LIN {X 0,Y 259.156,Z 1194.159,A -85,B 0,C 180,E1 -3.982,E2 -3.982} C_VEL
LIN {X 0,Y 240.249,Z 1207.459,A -85,B 0,C 180,E1 -6,E2 -6} C_VEL
LIN {X 0,Y 222.253,Z 1218.996,A -85,B 0,C 180,E1 -8.279,E2 -8.279} C_VEL
LIN {X 0,Y 202.836,Z 1230.338,A -85,B 0,C 180,E1 -11.248,E2 -11.248} C_VEL
LIN {X 0,Y 177.97,Z 1243.274,A -85,B 0,C 180,E1 -16.153,E2 -16.153} C_VEL
LIN {X 0,Y 159.555,Z 1251.828,A -85,B 0,C 180,E1 -21.01,E2 -21.01} C_VEL
LIN {X 0,Y 142.486,Z 1259.1,A -85,B 0,C 180,E1 -27.004,E2 -27.004} C_VEL
LIN {X 0,Y 125.055,Z 1266.027,A -85,B 0,C 180,E1 -35.71,E2 -35.71} C_VEL
LIN {X 0,Y 109.97,Z 1271.615,A -85,B 0,C 180,E1 -47.736,E2 -47.736} C_VEL
LIN {X 0,Y 101.633,Z 1274.813,A -85,B 0,C 180,E1 -59.251,E2 -59.251} C_VEL
LIN {X 0,Y 97.319,Z 1276.772,A -85,B 0,C 180,E1 -70.952,E2 -70.952} C_VEL
LIN {X 0,Y 95.995,Z 1277.735,A -85,B 0,C 180,E1 -81.701,E2 -81.701} C_VEL
LIN {X 0,Y 95.905,Z 1278.05,A -85,B 0,C 180,E1 -90.017,E2 -90.017} C_VEL
LIN {X 0,Y 95.996,Z 1277.726,A -85,B 0,C 180,E1 -98.402,E2 -98.402} C_VEL
LIN {X 0,Y 97.638,Z 1276.598,A -85,B 0,C 180,E1 -110.393,E2 -110.393} C_VEL
LIN {X 0,Y 104.256,Z 1273.841,A -85,B 0,C 180,E1 -125.148,E2 -125.148} C_VEL
LIN {X 0,Y 115.973,Z 1269.325,A -85,B 0,C 180,E1 -137.875,E2 -137.875} C_VEL
LIN {X 0,Y 129.201,Z 1264.301,A -85,B 0,C 180,E1 -146.72,E2 -146.72} C_VEL
LIN {X 0,Y 144.01,Z 1258.396,A -85,B 0,C 180,E1 -153.617,E2 -153.617} C_VEL
LIN {X 0,Y 161.221,Z 1251.006,A -85,B 0,C 180,E1 -159.494,E2 -159.494} C_VEL
LIN {X 0,Y 184.211,Z 1240.12,A -85,B 0,C 180,E1 -165.22,E2 -165.22} C_VEL
LIN {X 0,Y 204.707,Z 1229.147,A -85,B 0,C 180,E1 -169.075,E2 -169.075} C_VEL
LIN {X 0,Y 222.303,Z 1218.82,A -85,B 0,C 180,E1 -171.735,E2 -171.735} C_VEL
LIN {X 0,Y 240.473,Z 1207.142,A -85,B 0,C 180,E1 -174.033,E2 -174.033} C_VEL
LIN {X 0,Y 260.572,Z 1192.942,A -85,B 0,C 180,E1 -176.162,E2 -176.162} C_VEL
LIN {X 0,Y 283.358,Z 1174.812,A -85,B 0,C 180,E1 -178.18,E2 -178.18} C_VEL
LIN {X 0,Y 299.995,Z 1160.095,A -85,B 0,C 180,E1 -179.448,E2 -179.448} C_VEL
LIN {X 0,Y 311.22,Z 1149.435,A -85,B 0,C 180,E1 -180.208,E2 -180.208} C_VEL
LIN {X 0,Y 290.116,Z 1168.891,A -85,B 0,C 180,E1 -181.735,E2 -181.735} C_VEL
LIN {X 0,Y 272.413,Z 1183.527,A -85,B 0,C 180,E1 -183.212,E2 -183.212} C_VEL
LIN {X 0,Y 254.915,Z 1196.706,A -85,B 0,C 180,E1 -184.887,E2 -184.887} C_VEL
LIN {X 0,Y 236.716,Z 1209.198,A -85,B 0,C 180,E1 -186.921,E2 -186.921} C_VEL
LIN {X 0,Y 214.231,Z 1223.155,A -85,B 0,C 180,E1 -189.971,E2 -189.971} C_VEL
LIN {X 0,Y 192.466,Z 1235.016,A -85,B 0,C 180,E1 -193.689,E2 -193.689} C_VEL
LIN {X 0,Y 175.049,Z 1243.639,A -85,B 0,C 180,E1 -197.44,E2 -197.44} C_VEL
LIN {X 0,Y 157.697,Z 1251.486,A -85,B 0,C 180,E1 -202.201,E2 -202.201} C_VEL
LIN {X 0,Y 139.436,Z 1259.064,A -85,B 0,C 180,E1 -208.953,E2 -208.953} C_VEL
LIN {X 0,Y 121.037,Z 1265.976,A -85,B 0,C 180,E1 -219.037,E2 -219.037} C_VEL
LIN {X 0,Y 109.576,Z 1270.085,A -85,B 0,C 180,E1 -228.91,E2 -228.91} C_VEL
LIN {X 0,Y 101.75,Z 1272.968,A -85,B 0,C 180,E1 -239.905,E2 -239.905} C_VEL
LIN {X 0,Y 97.45,Z 1274.785,A -85,B 0,C 180,E1 -251.436,E2 -251.436} C_VEL
LIN {X 0,Y 96.054,Z 1275.667,A -85,B 0,C 180,E1 -262.206,E2 -262.206} C_VEL
LIN {X 0,Y 95.898,Z 1275.918,A -85,B 0,C 180,E1 -271.178,E2 -271.178} C_VEL
LIN {X 0,Y 96.228,Z 1275.57,A -85,B 0,C 180,E1 -280.762,E2 -280.762} C_VEL
LIN {X 0,Y 99.154,Z 1274.127,A -85,B 0,C 180,E1 -294.402,E2 -294.402} C_VEL
LIN {X 0,Y 107.15,Z 1271.002,A -85,B 0,C 180,E1 -308.384,E2 -308.384} C_VEL
LIN {X 0,Y 117.511,Z 1267.28,A -85,B 0,C 180,E1 -318.461,E2 -318.461} C_VEL
LIN {X 0,Y 130.322,Z 1262.576,A -85,B 0,C 180,E1 -326.724,E2 -326.724} C_VEL
LIN {X 0,Y 145.941,Z 1256.491,A -85,B 0,C 180,E1 -333.803,E2 -333.803} C_VEL
LIN {X 0,Y 166.537,Z 1247.783,A -85,B 0,C 180,E1 -340.461,E2 -340.461} C_VEL
LIN {X 0,Y 188.109,Z 1237.371,A -85,B 0,C 180,E1 -345.533,E2 -345.533} C_VEL
LIN {X 0,Y 206.779,Z 1227.428,A -85,B 0,C 180,E1 -348.941,E2 -348.941} C_VEL
LIN {X 0,Y 225.299,Z 1216.585,A -85,B 0,C 180,E1 -351.693,E2 -351.693} C_VEL
LIN {X 0,Y 247.131,Z 1202.487,A -85,B 0,C 180,E1 -354.353,E2 -354.353} C_VEL
LIN {X 0,Y 268.428,Z 1186.87,A -85,B 0,C 180,E1 -356.504,E2 -356.504} C_VEL
LIN {X 0,Y 286.095,Z 1172.556,A -85,B 0,C 180,E1 -358.03,E2 -358.03} C_VEL
LIN {X 0,Y 302.945,Z 1157.563,A -85,B 0,C 180,E1 -359.306,E2 -359.306} C_VEL
LIN {X 0,Y 310.594,Z 1150.361,A -85,B 0,C 180,E1 -359.845,E2 -359.845} C_VEL
LIN {X 0,Y 300.565,Z 1159.826,A -85,B 0,C 180,E1 -360.522,E2 -360.522} C_VEL
LIN {X 0,Y 294.883,Z 1165.108,A -85,B 0,C 180,E1 -360.731,E2 -360.731} C_VEL
LIN {X 0,Y 278.673,Z 1178.812,A -85,B 0,C 180,E1 -360.644,E2 -360.644} C_VEL
LIN {X 0,Y 273.535,Z 1182.795,A -85,B 0,C 180,E1 -360.881,E2 -360.881} C_VEL
LIN {X 0,Y 256.149,Z 1195.901,A -85,B 0,C 180,E1 -362.366,E2 -362.366} C_VEL
LIN {X 0,Y 238.547,Z 1208.008,A -85,B 0,C 180,E1 -364.111,E2 -364.111} C_VEL
LIN {X 0,Y 220.169,Z 1219.529,A -85,B 0,C 180,E1 -366.257,E2 -366.257} C_VEL
LIN {X 0,Y 197.647,Z 1232.322,A -85,B 0,C 180,E1 -369.493,E2 -369.493} C_VEL
LIN {X 0,Y 174.924,Z 1243.592,A -85,B 0,C 180,E1 -373.705,E2 -373.705} C_VEL
LIN {X 0,Y 156.208,Z 1251.959,A -85,B 0,C 180,E1 -378.279,E2 -378.279} C_VEL
LIN {X 0,Y 138.868,Z 1259.009,A -85,B 0,C 180,E1 -383.91,E2 -383.91} C_VEL
LIN {X 0,Y 120.629,Z 1265.829,A -85,B 0,C 180,E1 -392.307,E2 -392.307} C_VEL
LIN {X 0,Y 103.957,Z 1271.525,A -85,B 0,C 180,E1 -404.647,E2 -404.647} C_VEL
LIN {X 0,Y 94.627,Z 1274.723,A -85,B 0,C 180,E1 -416.692,E2 -416.692} C_VEL
LIN {X 0,Y 89.669,Z 1276.668,A -85,B 0,C 180,E1 -429.115,E2 -429.115} C_VEL
LIN {X 0,Y 88.018,Z 1277.644,A -85,B 0,C 180,E1 -440.868,E2 -440.868} C_VEL
LIN {X 0,Y 87.904,Z 1277.963,A -85,B 0,C 180,E1 -450.019,E2 -450.019} C_VEL
LIN {X 0,Y 88.019,Z 1277.638,A -85,B 0,C 180,E1 -459.17,E2 -459.17} C_VEL
LIN {X 0,Y 89.841,Z 1276.578,A -85,B 0,C 180,E1 -471.566,E2 -471.566} C_VEL
LIN {X 0,Y 96.126,Z 1274.204,A -85,B 0,C 180,E1 -485.772,E2 -485.772} C_VEL
LIN {X 0,Y 109.486,Z 1269.616,A -85,B 0,C 180,E1 -500.262,E2 -500.262} C_VEL
LIN {X 0,Y 124.095,Z 1264.466,A -85,B 0,C 180,E1 -509.58,E2 -509.58} C_VEL
LIN {X 0,Y 139.687,Z 1258.61,A -85,B 0,C 180,E1 -516.404,E2 -516.404} C_VEL
LIN {X 0,Y 156.776,Z 1251.627,A -85,B 0,C 180,E1 -521.885,E2 -521.885} C_VEL
LIN {X 0,Y 176.754,Z 1242.649,A -85,B 0,C 180,E1 -526.683,E2 -526.683} C_VEL
LIN {X 0,Y 201.696,Z 1229.933,A -85,B 0,C 180,E1 -531.16,E2 -531.16} C_VEL
LIN {X 0,Y 221.251,Z 1218.726,A -85,B 0,C 180,E1 -533.889,E2 -533.889} C_VEL
LIN {X 0,Y 239.573,Z 1207.163,A -85,B 0,C 180,E1 -536.006,E2 -536.006} C_VEL
LIN {X 0,Y 258.174,Z 1194.258,A -85,B 0,C 180,E1 -537.823,E2 -537.823} C_VEL
LIN {X 0,Y 280.988,Z 1176.612,A -85,B 0,C 180,E1 -539.696,E2 -539.696} C_VEL
LIN {X 0,Y 288.217,Z 1170.471,A -85,B 0,C 180,E1 -540.226,E2 -540.226} C_VEL
LIN {X 0,Y 271.084,Z 1184.386,A -85,B 0,C 180,E1 -541.547,E2 -541.547} C_VEL
LIN {X 0,Y 253.362,Z 1197.496,A -85,B 0,C 180,E1 -543.111,E2 -543.111} C_VEL
LIN {X 0,Y 232.002,Z 1211.815,A -85,B 0,C 180,E1 -545.348,E2 -545.348} C_VEL
LIN {X 0,Y 208.24,Z 1225.801,A -85,B 0,C 180,E1 -548.419,E2 -548.419} C_VEL
LIN {X 0,Y 189.744,Z 1235.564,A -85,B 0,C 180,E1 -551.402,E2 -551.402} C_VEL
LIN {X 0,Y 171.842,Z 1244.133,A -85,B 0,C 180,E1 -554.98,E2 -554.98} C_VEL
LIN {X 0,Y 153.065,Z 1252.278,A -85,B 0,C 180,E1 -559.812,E2 -559.812} C_VEL
LIN {X 0,Y 131.097,Z 1260.81,A -85,B 0,C 180,E1 -567.758,E2 -567.758} C_VEL
LIN {X 0,Y 114.712,Z 1266.474,A -85,B 0,C 180,E1 -576.666,E2 -576.666} C_VEL
LIN {X 0,Y 102.983,Z 1270.333,A -85,B 0,C 180,E1 -586.401,E2 -586.401} C_VEL
LIN {X 0,Y 94.394,Z 1273.169,A -85,B 0,C 180,E1 -598,E2 -598} C_VEL
LIN {X 0,Y 89.607,Z 1274.94,A -85,B 0,C 180,E1 -610.424,E2 -610.424} C_VEL
LIN {X 0,Y 88.053,Z 1275.777,A -85,B 0,C 180,E1 -622.15,E2 -622.15} C_VEL
LIN {X 0,Y 87.899,Z 1276.006,A -85,B 0,C 180,E1 -631.285,E2 -631.285} C_VEL
LIN {X 0,Y 88.245,Z 1275.68,A -85,B 0,C 180,E1 -641.086,E2 -641.086} C_VEL
LIN {X 0,Y 91.516,Z 1274.31,A -85,B 0,C 180,E1 -655.893,E2 -655.893} C_VEL
LIN {X 0,Y 100.534,Z 1271.182,A -85,B 0,C 180,E1 -671.003,E2 -671.003} C_VEL
LIN {X 0,Y 112.164,Z 1267.37,A -85,B 0,C 180,E1 -681.645,E2 -681.645} C_VEL
LIN {X 0,Y 126.259,Z 1262.549,A -85,B 0,C 180,E1 -690.071,E2 -690.071} C_VEL
LIN {X 0,Y 142.567,Z 1256.533,A -85,B 0,C 180,E1 -696.874,E2 -696.874} C_VEL
LIN {X 0,Y 163.922,Z 1247.874,A -85,B 0,C 180,E1 -703.224,E2 -703.224} C_VEL
LIN {X 0,Y 186.01,Z 1237.553,A -85,B 0,C 180,E1 -707.995,E2 -707.995} C_VEL
LIN {X 0,Y 205.337,Z 1227.518,A -85,B 0,C 180,E1 -711.235,E2 -711.235} C_VEL
LIN {X 0,Y 223.289,Z 1217.244,A -85,B 0,C 180,E1 -713.688,E2 -713.688} C_VEL
LIN {X 0,Y 242.557,Z 1205.1,A -85,B 0,C 180,E1 -715.888,E2 -715.888} C_VEL
LIN {X 0,Y 267.061,Z 1187.725,A -85,B 0,C 180,E1 -718.193,E2 -718.193} C_VEL
LIN {X 0,Y 284.932,Z 1173.485,A -85,B 0,C 180,E1 -719.615,E2 -719.615} C_VEL
LIN {X 0,Y 287.634,Z 1171.208,A -85,B 0,C 180,E1 -719.826,E2 -719.826} C_VEL
LIN {X 0,Y 273.535,Z 1182.795,A -85,B 0,C 180,E1 -720.881,E2 -720.881} C_VEL
LIN {X 0,Y 267.462,Z 1187.511,A -85,B 0,C 180,E1 -721.15,E2 -721.15} C_VEL
LIN {X 0,Y 250.268,Z 1199.952,A -85,B 0,C 180,E1 -721.16,E2 -721.16} C_VEL
LIN {X 0,Y 244.838,Z 1203.559,A -85,B 0,C 180,E1 -721.463,E2 -721.463} C_VEL
LIN {X 0,Y 223.382,Z 1217.085,A -85,B 0,C 180,E1 -723.621,E2 -723.621} C_VEL
LIN {X 0,Y 204.053,Z 1228.083,A -85,B 0,C 180,E1 -725.99,E2 -725.99} C_VEL
LIN {X 0,Y 184.206,Z 1238.279,A -85,B 0,C 180,E1 -728.992,E2 -728.992} C_VEL
LIN {X 0,Y 160.383,Z 1249.194,A -85,B 0,C 180,E1 -733.704,E2 -733.704} C_VEL
LIN {X 0,Y 138.962,Z 1257.691,A -85,B 0,C 180,E1 -739.551,E2 -739.551} C_VEL
LIN {X 0,Y 121.526,Z 1263.934,A -85,B 0,C 180,E1 -746.293,E2 -746.293} C_VEL
LIN {X 0,Y 105.71,Z 1269.123,A -85,B 0,C 180,E1 -755.239,E2 -755.239} C_VEL
LIN {X 0,Y 90.657,Z 1273.835,A -85,B 0,C 180,E1 -769.555,E2 -769.555} C_VEL
LIN {X 0,Y 82.633,Z 1276.386,A -85,B 0,C 180,E1 -785.167,E2 -785.167} C_VEL
LIN {X 0,Y 80.099,Z 1277.532,A -85,B 0,C 180,E1 -799.229,E2 -799.229} C_VEL
LIN {X 0,Y 79.896,Z 1277.863,A -85,B 0,C 180,E1 -809.304,E2 -809.304} C_VEL
LIN {X 0,Y 80.001,Z 1277.598,A -85,B 0,C 180,E1 -818.646,E2 -818.646} C_VEL
LIN {X 0,Y 81.557,Z 1276.77,A -85,B 0,C 180,E1 -830.847,E2 -830.847} C_VEL
LIN {X 0,Y 86.413,Z 1275.065,A -85,B 0,C 180,E1 -843.76,E2 -843.76} C_VEL
LIN {X 0,Y 95.914,Z 1272.105,A -85,B 0,C 180,E1 -856.525,E2 -856.525} C_VEL
LIN {X 0,Y 108.767,Z 1268.092,A -85,B 0,C 180,E1 -866.802,E2 -866.802} C_VEL
LIN {X 0,Y 126.154,Z 1262.31,A -85,B 0,C 180,E1 -875.737,E2 -875.737} C_VEL
LIN {X 0,Y 149.161,Z 1253.675,A -85,B 0,C 180,E1 -883.483,E2 -883.483} C_VEL
LIN {X 0,Y 168.619,Z 1245.417,A -85,B 0,C 180,E1 -888.112,E2 -888.112} C_VEL
LIN {X 0,Y 187.058,Z 1236.748,A -85,B 0,C 180,E1 -891.492,E2 -891.492} C_VEL
LIN {X 0,Y 206.022,Z 1226.885,A -85,B 0,C 180,E1 -894.281,E2 -894.281} C_VEL
LIN {X 0,Y 229.302,Z 1213.436,A -85,B 0,C 180,E1 -897.023,E2 -897.023} C_VEL
LIN {X 0,Y 252.014,Z 1198.391,A -85,B 0,C 180,E1 -899.182,E2 -899.182} C_VEL
LIN {X 0,Y 264.989,Z 1189.078,A -85,B 0,C 180,E1 -900.257,E2 -900.257} C_VEL
LIN {X 0,Y 242.172,Z 1204.967,A -85,B 0,C 180,E1 -902.219,E2 -902.219} C_VEL
LIN {X 0,Y 222.604,Z 1217.133,A -85,B 0,C 180,E1 -904.244,E2 -904.244} C_VEL
LIN {X 0,Y 204.315,Z 1227.427,A -85,B 0,C 180,E1 -906.513,E2 -906.513} C_VEL
LIN {X 0,Y 185.471,Z 1237.022,A -85,B 0,C 180,E1 -909.365,E2 -909.365} C_VEL
LIN {X 0,Y 162.144,Z 1247.681,A -85,B 0,C 180,E1 -913.916,E2 -913.916} C_VEL
LIN {X 0,Y 139.459,Z 1256.554,A -85,B 0,C 180,E1 -920.049,E2 -920.049} C_VEL
LIN {X 0,Y 122.809,Z 1262.407,A -85,B 0,C 180,E1 -926.39,E2 -926.39} C_VEL
LIN {X 0,Y 107.947,Z 1267.175,A -85,B 0,C 180,E1 -934.45,E2 -934.45} C_VEL
LIN {X 0,Y 95.035,Z 1271.05,A -85,B 0,C 180,E1 -945.155,E2 -945.155} C_VEL
LIN {X 0,Y 84.858,Z 1274.147,A -85,B 0,C 180,E1 -960.317,E2 -960.317} C_VEL
LIN {X 0,Y 80.485,Z 1275.717,A -85,B 0,C 180,E1 -976.326,E2 -976.326} C_VEL
LIN {X 0,Y 79.919,Z 1276.039,A -85,B 0,C 180,E1 -987.111,E2 -987.111} C_VEL
LIN {X 0,Y 79.987,Z 1275.939,A -85,B 0,C 180,E1 -996.439,E2 -996.439} C_VEL
LIN {X 0,Y 81.441,Z 1275.255,A -85,B 0,C 180,E1 -1009.337,E2 -1009.337} C_VEL
LIN {X 0,Y 86.743,Z 1273.528,A -85,B 0,C 180,E1 -1023.569,E2 -1023.569} C_VEL
LIN {X 0,Y 95.995,Z 1270.802,A -85,B 0,C 180,E1 -1035.92,E2 -1035.92} C_VEL
LIN {X 0,Y 108.508,Z 1267.054,A -85,B 0,C 180,E1 -1045.999,E2 -1045.999} C_VEL
LIN {X 0,Y 124.225,Z 1262.004,A -85,B 0,C 180,E1 -1054.318,E2 -1054.318} C_VEL
LIN {X 0,Y 146.064,Z 1254.251,A -85,B 0,C 180,E1 -1062.058,E2 -1062.058} C_VEL
LIN {X 0,Y 167.963,Z 1245.182,A -85,B 0,C 180,E1 -1067.443,E2 -1067.443} C_VEL
LIN {X 0,Y 187.239,Z 1236.278,A -85,B 0,C 180,E1 -1071.015,E2 -1071.015} C_VEL
LIN {X 0,Y 206.694,Z 1226.289,A -85,B 0,C 180,E1 -1073.891,E2 -1073.891} C_VEL
LIN {X 0,Y 230.321,Z 1212.76,A -85,B 0,C 180,E1 -1076.681,E2 -1076.681} C_VEL
LIN {X 0,Y 253.236,Z 1197.657,A -85,B 0,C 180,E1 -1078.869,E2 -1078.869} C_VEL
LIN {X 0,Y 264.571,Z 1189.623,A -85,B 0,C 180,E1 -1079.81,E2 -1079.81} C_VEL
LIN {X 0,Y 244.838,Z 1203.559,A -85,B 0,C 180,E1 -1081.463,E2 -1081.463} C_VEL
LIN {X 0,Y 238.395,Z 1207.737,A -85,B 0,C 180,E1 -1081.813,E2 -1081.813} C_VEL
LIN {X 0,Y 221.173,Z 1218.143,A -85,B 0,C 180,E1 -1081.931,E2 -1081.931} C_VEL
LIN {X 0,Y 214.631,Z 1221.892,A -85,B 0,C 180,E1 -1082.349,E2 -1082.349} C_VEL
LIN {X 0,Y 189.509,Z 1235.084,A -85,B 0,C 180,E1 -1085.45,E2 -1085.45} C_VEL
LIN {X 0,Y 169.841,Z 1244.228,A -85,B 0,C 180,E1 -1088.571,E2 -1088.571} C_VEL
LIN {X 0,Y 150.526,Z 1252.269,A -85,B 0,C 180,E1 -1092.518,E2 -1092.518} C_VEL
LIN {X 0,Y 130.389,Z 1259.747,A -85,B 0,C 180,E1 -1098.079,E2 -1098.079} C_VEL
LIN {X 0,Y 107.164,Z 1267.258,A -85,B 0,C 180,E1 -1107.809,E2 -1107.809} C_VEL
LIN {X 0,Y 91.737,Z 1271.681,A -85,B 0,C 180,E1 -1118.409,E2 -1118.409} C_VEL
LIN {X 0,Y 80.612,Z 1274.736,A -85,B 0,C 180,E1 -1131.392,E2 -1131.392} C_VEL
LIN {X 0,Y 74.378,Z 1276.56,A -85,B 0,C 180,E1 -1145.396,E2 -1145.396} C_VEL
LIN {X 0,Y 72.115,Z 1277.468,A -85,B 0,C 180,E1 -1158.831,E2 -1158.831} C_VEL
LIN {X 0,Y 71.896,Z 1277.775,A -85,B 0,C 180,E1 -1169.226,E2 -1169.226} C_VEL
LIN {X 0,Y 72.031,Z 1277.509,A -85,B 0,C 180,E1 -1179.612,E2 -1179.612} C_VEL
LIN {X 0,Y 74.024,Z 1276.663,A -85,B 0,C 180,E1 -1193.289,E2 -1193.289} C_VEL
LIN {X 0,Y 80.081,Z 1274.857,A -85,B 0,C 180,E1 -1207.745,E2 -1207.745} C_VEL
LIN {X 0,Y 90.63,Z 1271.946,A -85,B 0,C 180,E1 -1220.585,E2 -1220.585} C_VEL
LIN {X 0,Y 105.139,Z 1267.789,A -85,B 0,C 180,E1 -1231.064,E2 -1231.064} C_VEL
LIN {X 0,Y 126.244,Z 1261.179,A -85,B 0,C 180,E1 -1240.51,E2 -1240.51} C_VEL
LIN {X 0,Y 148.776,Z 1252.868,A -85,B 0,C 180,E1 -1247.073,E2 -1247.073} C_VEL
LIN {X 0,Y 168.021,Z 1244.915,A -85,B 0,C 180,E1 -1251.109,E2 -1251.109} C_VEL
LIN {X 0,Y 186.958,Z 1236.192,A -85,B 0,C 180,E1 -1254.195,E2 -1254.195} C_VEL
LIN {X 0,Y 207.31,Z 1225.754,A -85,B 0,C 180,E1 -1256.843,E2 -1256.843} C_VEL
LIN {X 0,Y 233.276,Z 1210.634,A -85,B 0,C 180,E1 -1259.509,E2 -1259.509} C_VEL
LIN {X 0,Y 241.697,Z 1205.247,A -85,B 0,C 180,E1 -1260.273,E2 -1260.273} C_VEL
LIN {X 0,Y 222.142,Z 1217.226,A -85,B 0,C 180,E1 -1262.095,E2 -1262.095} C_VEL
LIN {X 0,Y 202.996,Z 1227.804,A -85,B 0,C 180,E1 -1264.237,E2 -1264.237} C_VEL
LIN {X 0,Y 183.342,Z 1237.569,A -85,B 0,C 180,E1 -1266.937,E2 -1266.937} C_VEL
LIN {X 0,Y 159.07,Z 1248.271,A -85,B 0,C 180,E1 -1271.268,E2 -1271.268} C_VEL
LIN {X 0,Y 136.81,Z 1256.646,A -85,B 0,C 180,E1 -1276.747,E2 -1276.747} C_VEL
LIN {X 0,Y 119.33,Z 1262.499,A -85,B 0,C 180,E1 -1282.794,E2 -1282.794} C_VEL
LIN {X 0,Y 102.759,Z 1267.47,A -85,B 0,C 180,E1 -1291.072,E2 -1291.072} C_VEL
LIN {X 0,Y 87.523,Z 1271.657,A -85,B 0,C 180,E1 -1303.272,E2 -1303.272} C_VEL
LIN {X 0,Y 76.23,Z 1274.659,A -85,B 0,C 180,E1 -1320.943,E2 -1320.943} C_VEL
LIN {X 0,Y 72.367,Z 1275.868,A -85,B 0,C 180,E1 -1337.205,E2 -1337.205} C_VEL
LIN {X 0,Y 71.907,Z 1276.172,A -85,B 0,C 180,E1 -1348.383,E2 -1348.383} C_VEL
LIN {X 0,Y 72.085,Z 1275.984,A -85,B 0,C 180,E1 -1358.753,E2 -1358.753} C_VEL
LIN {X 0,Y 74.001,Z 1275.278,A -85,B 0,C 180,E1 -1372.205,E2 -1372.205} C_VEL
LIN {X 0,Y 80.096,Z 1273.595,A -85,B 0,C 180,E1 -1386.969,E2 -1386.969} C_VEL
LIN {X 0,Y 91.016,Z 1270.735,A -85,B 0,C 180,E1 -1400.233,E2 -1400.233} C_VEL
LIN {X 0,Y 105.514,Z 1266.738,A -85,B 0,C 180,E1 -1410.634,E2 -1410.634} C_VEL
LIN {X 0,Y 124.909,Z 1260.841,A -85,B 0,C 180,E1 -1419.44,E2 -1419.44} C_VEL
LIN {X 0,Y 148.13,Z 1252.598,A -85,B 0,C 180,E1 -1426.353,E2 -1426.353} C_VEL
LIN {X 0,Y 168.196,Z 1244.47,A -85,B 0,C 180,E1 -1430.615,E2 -1430.615} C_VEL
LIN {X 0,Y 187.068,Z 1235.914,A -85,B 0,C 180,E1 -1433.709,E2 -1433.709} C_VEL
LIN {X 0,Y 208.33,Z 1225.144,A -85,B 0,C 180,E1 -1436.485,E2 -1436.485} C_VEL
LIN {X 0,Y 233.961,Z 1210.327,A -85,B 0,C 180,E1 -1439.131,E2 -1439.131} C_VEL
LIN {X 0,Y 241.287,Z 1205.688,A -85,B 0,C 180,E1 -1439.793,E2 -1439.793} C_VEL
LIN {X 0,Y 222.019,Z 1217.572,A -85,B 0,C 180,E1 -1441.567,E2 -1441.567} C_VEL
LIN {X 0,Y 214.631,Z 1221.892,A -85,B 0,C 180,E1 -1442.349,E2 -1442.349} C_VEL
LIN {X 0,Y 208.006,Z 1225.581,A -85,B 0,C 180,E1 -1442.802,E2 -1442.802} C_VEL
LIN {X 0,Y 189.98,Z 1234.527,A -85,B 0,C 180,E1 -1443.095,E2 -1443.095} C_VEL
LIN {X 0,Y 183.148,Z 1237.712,A -85,B 0,C 180,E1 -1443.65,E2 -1443.65} C_VEL
LIN {X 0,Y 158.31,Z 1248.609,A -85,B 0,C 180,E1 -1447.527,E2 -1447.527} C_VEL
LIN {X 0,Y 134.272,Z 1257.509,A -85,B 0,C 180,E1 -1452.771,E2 -1452.771} C_VEL
LIN {X 0,Y 115.077,Z 1263.752,A -85,B 0,C 180,E1 -1458.774,E2 -1458.774} C_VEL
LIN {X 0,Y 97.494,Z 1268.811,A -85,B 0,C 180,E1 -1466.884,E2 -1466.884} C_VEL
LIN {X 0,Y 79.428,Z 1273.518,A -85,B 0,C 180,E1 -1480.982,E2 -1480.982} C_VEL
LIN {X 0,Y 68.189,Z 1276.189,A -85,B 0,C 180,E1 -1499.151,E2 -1499.151} C_VEL
LIN {X 0,Y 64.268,Z 1277.355,A -85,B 0,C 180,E1 -1516.531,E2 -1516.531} C_VEL
LIN {X 0,Y 63.899,Z 1277.665,A -85,B 0,C 180,E1 -1528.233,E2 -1528.233} C_VEL
LIN {X 0,Y 64.008,Z 1277.469,A -85,B 0,C 180,E1 -1539.013,E2 -1539.013} C_VEL
LIN {X 0,Y 66.07,Z 1276.732,A -85,B 0,C 180,E1 -1554.144,E2 -1554.144} C_VEL
LIN {X 0,Y 72.801,Z 1275,A -85,B 0,C 180,E1 -1570.232,E2 -1570.232} C_VEL
LIN {X 0,Y 84.935,Z 1272.017,A -85,B 0,C 180,E1 -1584.35,E2 -1584.35} C_VEL
LIN {X 0,Y 100.578,Z 1267.907,A -85,B 0,C 180,E1 -1594.812,E2 -1594.812} C_VEL
LIN {X 0,Y 120.228,Z 1262.125,A -85,B 0,C 180,E1 -1603.059,E2 -1603.059} C_VEL
LIN {X 0,Y 145.271,Z 1253.489,A -85,B 0,C 180,E1 -1609.87,E2 -1609.87} C_VEL
LIN {X 0,Y 165.971,Z 1245.23,A -85,B 0,C 180,E1 -1613.807,E2 -1613.807} C_VEL
LIN {X 0,Y 185.317,Z 1236.561,A -85,B 0,C 180,E1 -1616.643,E2 -1616.643} C_VEL
LIN {X 0,Y 205.03,Z 1226.697,A -85,B 0,C 180,E1 -1618.959,E2 -1618.959} C_VEL
LIN {X 0,Y 218.121,Z 1219.526,A -85,B 0,C 180,E1 -1620.298,E2 -1620.298} C_VEL
LIN {X 0,Y 193.254,Z 1232.661,A -85,B 0,C 180,E1 -1622.951,E2 -1622.951} C_VEL
LIN {X 0,Y 169.982,Z 1243.21,A -85,B 0,C 180,E1 -1626.156,E2 -1626.156} C_VEL
LIN {X 0,Y 150.165,Z 1251.159,A -85,B 0,C 180,E1 -1629.73,E2 -1629.73} C_VEL
LIN {X 0,Y 131.068,Z 1257.937,A -85,B 0,C 180,E1 -1634.296,E2 -1634.296} C_VEL
LIN {X 0,Y 110.532,Z 1264.347,A -85,B 0,C 180,E1 -1641.256,E2 -1641.256} C_VEL
LIN {X 0,Y 88.673,Z 1270.137,A -85,B 0,C 180,E1 -1653.414,E2 -1653.414} C_VEL
LIN {X 0,Y 75.244,Z 1273.292,A -85,B 0,C 180,E1 -1666.961,E2 -1666.961} C_VEL
LIN {X 0,Y 67.6,Z 1275.077,A -85,B 0,C 180,E1 -1681.724,E2 -1681.724} C_VEL
LIN {X 0,Y 64.327,Z 1275.999,A -85,B 0,C 180,E1 -1697.405,E2 -1697.405} C_VEL
LIN {X 0,Y 63.907,Z 1276.302,A -85,B 0,C 180,E1 -1709.974,E2 -1709.974} C_VEL
LIN {X 0,Y 64.318,Z 1276.008,A -85,B 0,C 180,E1 -1722.544,E2 -1722.544} C_VEL
LIN {X 0,Y 67.847,Z 1275.039,A -85,B 0,C 180,E1 -1739.071,E2 -1739.071} C_VEL
LIN {X 0,Y 77.083,Z 1272.926,A -85,B 0,C 180,E1 -1755.535,E2 -1755.535} C_VEL
LIN {X 0,Y 95.187,Z 1268.581,A -85,B 0,C 180,E1 -1771.105,E2 -1771.105} C_VEL
LIN {X 0,Y 113.739,Z 1263.44,A -85,B 0,C 180,E1 -1780.11,E2 -1780.11} C_VEL
LIN {X 0,Y 132.753,Z 1257.452,A -85,B 0,C 180,E1 -1786.254,E2 -1786.254} C_VEL
LIN {X 0,Y 152.872,Z 1250.243,A -85,B 0,C 180,E1 -1790.899,E2 -1790.899} C_VEL
LIN {X 0,Y 177.602,Z 1240.099,A -85,B 0,C 180,E1 -1795.062,E2 -1795.062} C_VEL
LIN {X 0,Y 201.057,Z 1228.81,A -85,B 0,C 180,E1 -1798.042,E2 -1798.042} C_VEL
LIN {X 0,Y 217.938,Z 1219.79,A -85,B 0,C 180,E1 -1799.769,E2 -1799.769} C_VEL
LIN {X 0,Y 193.109,Z 1233.009,A -85,B 0,C 180,E1 -1802.393,E2 -1802.393} C_VEL
LIN {X 0,Y 183.148,Z 1237.712,A -85,B 0,C 180,E1 -1803.65,E2 -1803.65} C_VEL
LIN {X 0,Y 176.292,Z 1240.91,A -85,B 0,C 180,E1 -1804.252,E2 -1804.252} C_VEL
LIN {X 0,Y 156.677,Z 1248.828,A -85,B 0,C 180,E1 -1804.904,E2 -1804.904} C_VEL
LIN {X 0,Y 150.703,Z 1251.005,A -85,B 0,C 180,E1 -1805.614,E2 -1805.614} C_VEL
LIN {X 0,Y 130.656,Z 1258.08,A -85,B 0,C 180,E1 -1809.693,E2 -1809.693} C_VEL
LIN {X 0,Y 110.893,Z 1264.177,A -85,B 0,C 180,E1 -1815.316,E2 -1815.316} C_VEL
LIN {X 0,Y 88.179,Z 1270.246,A -85,B 0,C 180,E1 -1825.524,E2 -1825.524} C_VEL
LIN {X 0,Y 70.546,Z 1274.129,A -85,B 0,C 180,E1 -1840.1,E2 -1840.1} C_VEL
LIN {X 0,Y 60.552,Z 1276.24,A -85,B 0,C 180,E1 -1857.014,E2 -1857.014} C_VEL
LIN {X 0,Y 56.319,Z 1277.291,A -85,B 0,C 180,E1 -1875.639,E2 -1875.639} C_VEL
LIN {X 0,Y 55.896,Z 1277.6,A -85,B 0,C 180,E1 -1889.005,E2 -1889.005} C_VEL
LIN {X 0,Y 56.108,Z 1277.354,A -85,B 0,C 180,E1 -1901.433,E2 -1901.433} C_VEL
LIN {X 0,Y 58.973,Z 1276.571,A -85,B 0,C 180,E1 -1918.373,E2 -1918.373} C_VEL
LIN {X 0,Y 67.363,Z 1274.764,A -85,B 0,C 180,E1 -1935.763,E2 -1935.763} C_VEL
LIN {X 0,Y 80.758,Z 1271.834,A -85,B 0,C 180,E1 -1949.494,E2 -1949.494} C_VEL
LIN {X 0,Y 97.305,Z 1267.815,A -85,B 0,C 180,E1 -1959.285,E2 -1959.285} C_VEL
LIN {X 0,Y 118.053,Z 1262.032,A -85,B 0,C 180,E1 -1966.963,E2 -1966.963} C_VEL
LIN {X 0,Y 144.397,Z 1253.257,A -85,B 0,C 180,E1 -1973.24,E2 -1973.24} C_VEL
LIN {X 0,Y 165.275,Z 1245.137,A -85,B 0,C 180,E1 -1976.707,E2 -1976.707} C_VEL
LIN {X 0,Y 185.015,Z 1236.467,A -85,B 0,C 180,E1 -1979.244,E2 -1979.244} C_VEL
LIN {X 0,Y 194.661,Z 1231.966,A -85,B 0,C 180,E1 -1980.294,E2 -1980.294} C_VEL
LIN {X 0,Y 169.289,Z 1243.303,A -85,B 0,C 180,E1 -1983.338,E2 -1983.338} C_VEL
LIN {X 0,Y 148.975,Z 1251.253,A -85,B 0,C 180,E1 -1986.552,E2 -1986.552} C_VEL
LIN {X 0,Y 129.196,Z 1258.048,A -85,B 0,C 180,E1 -1990.705,E2 -1990.705} C_VEL
LIN {X 0,Y 107.785,Z 1264.439,A -85,B 0,C 180,E1 -1997.114,E2 -1997.114} C_VEL
LIN {X 0,Y 84.378,Z 1270.228,A -85,B 0,C 180,E1 -2008.693,E2 -2008.693} C_VEL
LIN {X 0,Y 69.825,Z 1273.309,A -85,B 0,C 180,E1 -2021.84,E2 -2021.84} C_VEL
LIN {X 0,Y 60.52,Z 1275.167,A -85,B 0,C 180,E1 -2038.053,E2 -2038.053} C_VEL
LIN {X 0,Y 56.462,Z 1276.088,A -85,B 0,C 180,E1 -2055.616,E2 -2055.616} C_VEL
LIN {X 0,Y 55.904,Z 1276.369,A -85,B 0,C 180,E1 -2068.946,E2 -2068.946} C_VEL
LIN {X 0,Y 56.269,Z 1276.14,A -85,B 0,C 180,E1 -2082.217,E2 -2082.217} C_VEL
LIN {X 0,Y 59.507,Z 1275.391,A -85,B 0,C 180,E1 -2099.129,E2 -2099.129} C_VEL
LIN {X 0,Y 68.082,Z 1273.687,A -85,B 0,C 180,E1 -2115.987,E2 -2115.987} C_VEL
LIN {X 0,Y 81.394,Z 1270.916,A -85,B 0,C 180,E1 -2129.263,E2 -2129.263} C_VEL
LIN {X 0,Y 98.545,Z 1266.885,A -85,B 0,C 180,E1 -2139.199,E2 -2139.199} C_VEL
LIN {X 0,Y 121.863,Z 1260.52,A -85,B 0,C 180,E1 -2147.452,E2 -2147.452} C_VEL
LIN {X 0,Y 146.039,Z 1252.43,A -85,B 0,C 180,E1 -2152.991,E2 -2152.991} C_VEL
LIN {X 0,Y 166.286,Z 1244.651,A -85,B 0,C 180,E1 -2156.327,E2 -2156.327} C_VEL
LIN {X 0,Y 185.979,Z 1236.094,A -85,B 0,C 180,E1 -2158.847,E2 -2158.847} C_VEL
LIN {X 0,Y 194.324,Z 1232.273,A -85,B 0,C 180,E1 -2159.753,E2 -2159.753} C_VEL
LIN {X 0,Y 169.14,Z 1243.638,A -85,B 0,C 180,E1 -2162.757,E2 -2162.757} C_VEL
LIN {X 0,Y 150.703,Z 1251.005,A -85,B 0,C 180,E1 -2165.614,E2 -2165.614} C_VEL
LIN {X 0,Y 143.693,Z 1253.574,A -85,B 0,C 180,E1 -2166.469,E2 -2166.469} C_VEL
LIN {X 0,Y 123.627,Z 1259.975,A -85,B 0,C 180,E1 -2167.663,E2 -2167.663} C_VEL
LIN {X 0,Y 117.586,Z 1261.694,A -85,B 0,C 180,E1 -2168.715,E2 -2168.715} C_VEL
LIN {X 0,Y 95.49,Z 1267.579,A -85,B 0,C 180,E1 -2175.634,E2 -2175.634} C_VEL
LIN {X 0,Y 77.94,Z 1271.56,A -85,B 0,C 180,E1 -2184.433,E2 -2184.433} C_VEL
LIN {X 0,Y 63.491,Z 1274.4,A -85,B 0,C 180,E1 -2196.758,E2 -2196.758} C_VEL
LIN {X 0,Y 53.023,Z 1276.292,A -85,B 0,C 180,E1 -2214.267,E2 -2214.267} C_VEL
LIN {X 0,Y 48.388,Z 1277.227,A -85,B 0,C 180,E1 -2234.453,E2 -2234.453} C_VEL
LIN {X 0,Y 47.896,Z 1277.513,A -85,B 0,C 180,E1 -2248.838,E2 -2248.838} C_VEL
LIN {X 0,Y 48.16,Z 1277.28,A -85,B 0,C 180,E1 -2262.628,E2 -2262.628} C_VEL
LIN {X 0,Y 51.566,Z 1276.552,A -85,B 0,C 180,E1 -2281.606,E2 -2281.606} C_VEL
LIN {X 0,Y 61.239,Z 1274.795,A -85,B 0,C 180,E1 -2300.448,E2 -2300.448} C_VEL
LIN {X 0,Y 75.963,Z 1271.931,A -85,B 0,C 180,E1 -2314.254,E2 -2314.254} C_VEL
LIN {X 0,Y 93.792,Z 1267.932,A -85,B 0,C 180,E1 -2323.684,E2 -2323.684} C_VEL
LIN {X 0,Y 114.257,Z 1262.544,A -85,B 0,C 180,E1 -2330.429,E2 -2330.429} C_VEL
LIN {X 0,Y 140.345,Z 1254.373,A -85,B 0,C 180,E1 -2336.019,E2 -2336.019} C_VEL
LIN {X 0,Y 164.009,Z 1245.452,A -85,B 0,C 180,E1 -2339.502,E2 -2339.502} C_VEL
LIN {X 0,Y 170.439,Z 1242.82,A -85,B 0,C 180,E1 -2340.336,E2 -2340.336} C_VEL
LIN {X 0,Y 149.235,Z 1250.995,A -85,B 0,C 180,E1 -2343.182,E2 -2343.182} C_VEL
LIN {X 0,Y 128.915,Z 1257.823,A -85,B 0,C 180,E1 -2346.8,E2 -2346.8} C_VEL
LIN {X 0,Y 108.356,Z 1263.779,A -85,B 0,C 180,E1 -2351.94,E2 -2351.94} C_VEL
LIN {X 0,Y 84.026,Z 1269.681,A -85,B 0,C 180,E1 -2361.647,E2 -2361.647} C_VEL
LIN {X 0,Y 65.254,Z 1273.289,A -85,B 0,C 180,E1 -2375.656,E2 -2375.656} C_VEL
LIN {X 0,Y 53.751,Z 1275.256,A -85,B 0,C 180,E1 -2393.432,E2 -2393.432} C_VEL
LIN {X 0,Y 48.665,Z 1276.176,A -85,B 0,C 180,E1 -2413.248,E2 -2413.248} C_VEL
LIN {X 0,Y 47.905,Z 1276.457,A -85,B 0,C 180,E1 -2428.77,E2 -2428.77} C_VEL
LIN {X 0,Y 48.345,Z 1276.24,A -85,B 0,C 180,E1 -2443.569,E2 -2443.569} C_VEL
LIN {X 0,Y 52.185,Z 1275.539,A -85,B 0,C 180,E1 -2462.534,E2 -2462.534} C_VEL
LIN {X 0,Y 62.015,Z 1273.887,A -85,B 0,C 180,E1 -2480.662,E2 -2480.662} C_VEL
LIN {X 0,Y 76.699,Z 1271.163,A -85,B 0,C 180,E1 -2494.04,E2 -2494.04} C_VEL
LIN {X 0,Y 94.897,Z 1267.209,A -85,B 0,C 180,E1 -2503.472,E2 -2503.472} C_VEL
LIN {X 0,Y 115.645,Z 1261.866,A -85,B 0,C 180,E1 -2510.186,E2 -2510.186} C_VEL
LIN {X 0,Y 143.622,Z 1253.106,A -85,B 0,C 180,E1 -2516.008,E2 -2516.008} C_VEL
LIN {X 0,Y 165.96,Z 1244.741,A -85,B 0,C 180,E1 -2519.215,E2 -2519.215} C_VEL
LIN {X 0,Y 170.341,Z 1242.977,A -85,B 0,C 180,E1 -2519.737,E2 -2519.737} C_VEL
LIN {X 0,Y 149.097,Z 1251.282,A -85,B 0,C 180,E1 -2522.564,E2 -2522.564} C_VEL
LIN {X 0,Y 128.337,Z 1258.363,A -85,B 0,C 180,E1 -2526.262,E2 -2526.262} C_VEL
LIN {X 0,Y 117.586,Z 1261.694,A -85,B 0,C 180,E1 -2528.715,E2 -2528.715} C_VEL
LIN {X 0,Y 110.513,Z 1263.625,A -85,B 0,C 180,E1 -2530.029,E2 -2530.029} C_VEL
LIN {X 0,Y 90.205,Z 1268.341,A -85,B 0,C 180,E1 -2532.411,E2 -2532.411} C_VEL
LIN {X 0,Y 84.253,Z 1269.644,A -85,B 0,C 180,E1 -2534.165,E2 -2534.165} C_VEL
LIN {X 0,Y 61.193,Z 1273.948,A -85,B 0,C 180,E1 -2548.135,E2 -2548.135} C_VEL
LIN {X 0,Y 47.11,Z 1276.132,A -85,B 0,C 180,E1 -2567.27,E2 -2567.27} C_VEL
LIN {X 0,Y 40.818,Z 1277.114,A -85,B 0,C 180,E1 -2589.987,E2 -2589.987} C_VEL
LIN {X 0,Y 39.895,Z 1277.425,A -85,B 0,C 180,E1 -2608.605,E2 -2608.605} C_VEL
LIN {X 0,Y 40.249,Z 1277.204,A -85,B 0,C 180,E1 -2624.426,E2 -2624.426} C_VEL
LIN {X 0,Y 44.793,Z 1276.462,A -85,B 0,C 180,E1 -2647.108,E2 -2647.108} C_VEL
LIN {X 0,Y 56.186,Z 1274.727,A -85,B 0,C 180,E1 -2666.813,E2 -2666.813} C_VEL
LIN {X 0,Y 72.388,Z 1271.905,A -85,B 0,C 180,E1 -2679.989,E2 -2679.989} C_VEL
LIN {X 0,Y 90.872,Z 1268.05,A -85,B 0,C 180,E1 -2688.395,E2 -2688.395} C_VEL
LIN {X 0,Y 110.608,Z 1263.136,A -85,B 0,C 180,E1 -2694.048,E2 -2694.048} C_VEL
LIN {X 0,Y 132.255,Z 1256.767,A -85,B 0,C 180,E1 -2698.267,E2 -2698.267} C_VEL
LIN {X 0,Y 146.24,Z 1252.055,A -85,B 0,C 180,E1 -2700.324,E2 -2700.324} C_VEL
LIN {X 0,Y 123.305,Z 1259.413,A -85,B 0,C 180,E1 -2703.968,E2 -2703.968} C_VEL
LIN {X 0,Y 95.687,Z 1266.62,A -85,B 0,C 180,E1 -2710.73,E2 -2710.73} C_VEL
LIN {X 0,Y 75.205,Z 1270.881,A -85,B 0,C 180,E1 -2719.21,E2 -2719.21} C_VEL
LIN {X 0,Y 58.621,Z 1273.712,A -85,B 0,C 180,E1 -2731.428,E2 -2731.428} C_VEL
LIN {X 0,Y 46.433,Z 1275.478,A -85,B 0,C 180,E1 -2749.714,E2 -2749.714} C_VEL
LIN {X 0,Y 40.796,Z 1276.286,A -85,B 0,C 180,E1 -2771.379,E2 -2771.379} C_VEL
LIN {X 0,Y 39.905,Z 1276.545,A -85,B 0,C 180,E1 -2788.523,E2 -2788.523} C_VEL
LIN {X 0,Y 40.457,Z 1276.34,A -85,B 0,C 180,E1 -2805.447,E2 -2805.447} C_VEL
LIN {X 0,Y 45.455,Z 1275.635,A -85,B 0,C 180,E1 -2827.971,E2 -2827.971} C_VEL
LIN {X 0,Y 57.297,Z 1273.952,A -85,B 0,C 180,E1 -2847.249,E2 -2847.249} C_VEL
LIN {X 0,Y 73.438,Z 1271.254,A -85,B 0,C 180,E1 -2859.889,E2 -2859.889} C_VEL
LIN {X 0,Y 91.932,Z 1267.507,A -85,B 0,C 180,E1 -2868.101,E2 -2868.101} C_VEL
LIN {X 0,Y 112.593,Z 1262.458,A -85,B 0,C 180,E1 -2873.892,E2 -2873.892} C_VEL
LIN {X 0,Y 138.983,Z 1254.708,A -85,B 0,C 180,E1 -2878.731,E2 -2878.731} C_VEL
LIN {X 0,Y 145.95,Z 1252.262,A -85,B 0,C 180,E1 -2879.72,E2 -2879.72} C_VEL
LIN {X 0,Y 120.228,Z 1260.609,A -85,B 0,C 180,E1 -2883.885,E2 -2883.885} C_VEL
LIN {X 0,Y 94.503,Z 1267.278,A -85,B 0,C 180,E1 -2890.381,E2 -2890.381} C_VEL
LIN {X 0,Y 84.253,Z 1269.644,A -85,B 0,C 180,E1 -2894.165,E2 -2894.165} C_VEL
LIN {X 0,Y 77.332,Z 1271.058,A -85,B 0,C 180,E1 -2896.452,E2 -2896.452} C_VEL
LIN {X 0,Y 56.795,Z 1274.041,A -85,B 0,C 180,E1 -2902.347,E2 -2902.347} C_VEL
LIN {X 0,Y 51.724,Z 1274.725,A -85,B 0,C 180,E1 -2905.906,E2 -2905.906} C_VEL
LIN {X 0,Y 36.101,Z 1276.747,A -85,B 0,C 180,E1 -2932.518,E2 -2932.518} C_VEL
LIN {X 0,Y 31.942,Z 1277.268,A -85,B 0,C 180,E1 -2962.859,E2 -2962.859} C_VEL
LIN {X 0,Y 31.944,Z 1277.26,A -85,B 0,C 180,E1 -2977.244,E2 -2977.244} C_VEL
LIN {X 0,Y 36.125,Z 1276.725,A -85,B 0,C 180,E1 -3007.567,E2 -3007.567} C_VEL
LIN {X 0,Y 51.33,Z 1274.752,A -85,B 0,C 180,E1 -3033.711,E2 -3033.711} C_VEL
LIN {X 0,Y 69.973,Z 1271.813,A -85,B 0,C 180,E1 -3046.424,E2 -3046.424} C_VEL
LIN {X 0,Y 89.563,Z 1267.957,A -85,B 0,C 180,E1 -3053.658,E2 -3053.658} C_VEL
LIN {X 0,Y 111.044,Z 1262.785,A -85,B 0,C 180,E1 -3058.595,E2 -3058.595} C_VEL
LIN {X 0,Y 121.279,Z 1260.024,A -85,B 0,C 180,E1 -3060.341,E2 -3060.341} C_VEL
LIN {X 0,Y 94.488,Z 1266.712,A -85,B 0,C 180,E1 -3065.744,E2 -3065.744} C_VEL
LIN {X 0,Y 73.802,Z 1270.816,A -85,B 0,C 180,E1 -3072.625,E2 -3072.625} C_VEL
LIN {X 0,Y 55.571,Z 1273.693,A -85,B 0,C 180,E1 -3083.348,E2 -3083.348} C_VEL
LIN {X 0,Y 41.137,Z 1275.502,A -85,B 0,C 180,E1 -3101.048,E2 -3101.048} C_VEL
LIN {X 0,Y 33.226,Z 1276.374,A -85,B 0,C 180,E1 -3126.917,E2 -3126.917} C_VEL
LIN {X 0,Y 31.905,Z 1276.632,A -85,B 0,C 180,E1 -3148.152,E2 -3148.152} C_VEL
LIN {X 0,Y 32.622,Z 1276.442,A -85,B 0,C 180,E1 -3168.162,E2 -3168.162} C_VEL
LIN {X 0,Y 38.778,Z 1275.79,A -85,B 0,C 180,E1 -3194.06,E2 -3194.06} C_VEL
LIN {X 0,Y 53.098,Z 1274.067,A -85,B 0,C 180,E1 -3214.596,E2 -3214.596} C_VEL
LIN {X 0,Y 71.007,Z 1271.344,A -85,B 0,C 180,E1 -3226.209,E2 -3226.209} C_VEL
LIN {X 0,Y 90.579,Z 1267.598,A -85,B 0,C 180,E1 -3233.283,E2 -3233.283} C_VEL
LIN {X 0,Y 112.011,Z 1262.549,A -85,B 0,C 180,E1 -3238.154,E2 -3238.154} C_VEL
LIN {X 0,Y 120.953,Z 1260.211,A -85,B 0,C 180,E1 -3239.715,E2 -3239.715} C_VEL
LIN {X 0,Y 94.324,Z 1266.977,A -85,B 0,C 180,E1 -3245.064,E2 -3245.064} C_VEL
LIN {X 0,Y 73.556,Z 1271.215,A -85,B 0,C 180,E1 -3251.958,E2 -3251.958} C_VEL
LIN {X 0,Y 55.268,Z 1274.208,A -85,B 0,C 180,E1 -3262.763,E2 -3262.763} C_VEL
LIN {X 0,Y 51.724,Z 1274.725,A -85,B 0,C 180,E1 -3265.906,E2 -3265.906} C_VEL
LIN {X 0,Y 45.499,Z 1275.542,A -85,B 0,C 180,E1 -3271.293,E2 -3271.293} C_VEL
LIN {X 0,Y 31.934,Z 1276.658,A -85,B 0,C 180,E1 -3284.683,E2 -3284.683} C_VEL
LIN {X 0,Y 25.946,Z 1276.965,A -85,B 0,C 180,E1 -3299.482,E2 -3299.482} C_VEL
LIN {X 0,Y 25.145,Z 1277.01,A -85,B 0,C 180,E1 -3304.176,E2 -3304.176} C_VEL
LIN {X 0,Y 23.9,Z 1277.262,A -85,B 0,C 180,E1 -3330.069,E2 -3330.069} C_VEL
LIN {X 0,Y 25.47,Z 1276.978,A -85,B 0,C 180,E1 -3358.178,E2 -3358.178} C_VEL
LIN {X 0,Y 36.056,Z 1276,A -85,B 0,C 180,E1 -3389.365,E2 -3389.365} C_VEL
LIN {X 0,Y 53.571,Z 1273.962,A -85,B 0,C 180,E1 -3406.181,E2 -3406.181} C_VEL
LIN {X 0,Y 77.201,Z 1270.254,A -85,B 0,C 180,E1 -3416.043,E2 -3416.043} C_VEL
LIN {X 0,Y 95.599,Z 1266.482,A -85,B 0,C 180,E1 -3420.361,E2 -3420.361} C_VEL
LIN {X 0,Y 72.439,Z 1270.908,A -85,B 0,C 180,E1 -3426.187,E2 -3426.187} C_VEL
LIN {X 0,Y 52.841,Z 1273.784,A -85,B 0,C 180,E1 -3435.083,E2 -3435.083} C_VEL
LIN {X 0,Y 35.699,Z 1275.644,A -85,B 0,C 180,E1 -3452.153,E2 -3452.153} C_VEL
LIN {X 0,Y 25.624,Z 1276.484,A -85,B 0,C 180,E1 -3482.007,E2 -3482.007} C_VEL
LIN {X 0,Y 23.904,Z 1276.739,A -85,B 0,C 180,E1 -3509.931,E2 -3509.931} C_VEL
LIN {X 0,Y 25.594,Z 1276.492,A -85,B 0,C 180,E1 -3537.883,E2 -3537.883} C_VEL
LIN {X 0,Y 35.55,Z 1275.677,A -85,B 0,C 180,E1 -3567.696,E2 -3567.696} C_VEL
LIN {X 0,Y 51.878,Z 1273.936,A -85,B 0,C 180,E1 -3584.385,E2 -3584.385} C_VEL
LIN {X 0,Y 71.46,Z 1271.114,A -85,B 0,C 180,E1 -3593.573,E2 -3593.573} C_VEL
LIN {X 0,Y 92.965,Z 1267.079,A -85,B 0,C 180,E1 -3599.204,E2 -3599.204} C_VEL
LIN {X 0,Y 95.391,Z 1266.584,A -85,B 0,C 180,E1 -3599.682,E2 -3599.682} C_VEL
LIN {X 0,Y 71.926,Z 1271.185,A -85,B 0,C 180,E1 -3605.584,E2 -3605.584} C_VEL
LIN {X 0,Y 51.72,Z 1274.234,A -85,B 0,C 180,E1 -3614.976,E2 -3614.976} C_VEL
LIN {X 0,Y 35.287,Z 1276.094,A -85,B 0,C 180,E1 -3631.872,E2 -3631.872} C_VEL
LIN {X 0,Y 25.453,Z 1276.985,A -85,B 0,C 180,E1 -3661.949,E2 -3661.949} C_VEL
LIN {X 0,Y 25.145,Z 1277.01,A -85,B 0,C 180,E1 -3664.176,E2 -3664.176} C_VEL
LIN {X 0,Y 23.144,Z 1277.161,A -85,B 0,C 180,E1 -3677.779,E2 -3677.779} C_VEL
LIN {X 0,Y 20.704,Z 1277.193,A -85,B 0,C 180,E1 -3697.286,E2 -3697.286} C_VEL
LIN {X 0,Y 23.793,Z 1276.684,A -85,B 0,C 180,E1 -3747.202,E2 -3747.202} C_VEL
LIN {X 0,Y 26.214,Z 1276.453,A -85,B 0,C 180,E1 -3752.858,E2 -3752.858} C_VEL
LIN {X 0,Y 46.952,Z 1274.507,A -85,B 0,C 180,E1 -3772.659,E2 -3772.659} C_VEL
LIN {X 0,Y 68.645,Z 1271.527,A -85,B 0,C 180,E1 -3780.389,E2 -3780.389} C_VEL
LIN {X 0,Y 47.474,Z 1274.317,A -85,B 0,C 180,E1 -3787.923,E2 -3787.923} C_VEL
LIN {X 0,Y 26.932,Z 1276.141,A -85,B 0,C 180,E1 -3806.867,E2 -3806.867} C_VEL
LIN {X 0,Y 16.349,Z 1276.72,A -85,B 0,C 180,E1 -3852.089,E2 -3852.089} C_VEL
LIN {X 0,Y 16.037,Z 1276.771,A -85,B 0,C 180,E1 -3880.675,E2 -3880.675} C_VEL
LIN {X 0,Y 24.566,Z 1276.363,A -85,B 0,C 180,E1 -3928.6,E2 -3928.6} C_VEL
LIN {X 0,Y 46.458,Z 1274.469,A -85,B 0,C 180,E1 -3951.633,E2 -3951.633} C_VEL
LIN {X 0,Y 68.482,Z 1271.6,A -85,B 0,C 180,E1 -3959.655,E2 -3959.655} C_VEL
LIN {X 0,Y 45.423,Z 1274.727,A -85,B 0,C 180,E1 -3968.15,E2 -3968.15} C_VEL
LIN {X 0,Y 22.953,Z 1276.722,A -85,B 0,C 180,E1 -3994.271,E2 -3994.271} C_VEL
LIN {X 0,Y 15.924,Z 1277.139,A -85,B 0,C 180,E1 -4042.89,E2 -4042.89} C_VEL
LIN {X 0,Y 16.456,Z 1277.036,A -85,B 0,C 180,E1 -4071.488,E2 -4071.488} C_VEL
LIN {X 0,Y 26.214,Z 1276.453,A -85,B 0,C 180,E1 -4112.858,E2 -4112.858} C_VEL
LIN {X 0,Y 26.473,Z 1276.373,A -85,B 0,C 180,E1 -4116.614,E2 -4116.614} C_VEL
LIN {X 0,Y 24.756,Z 1276.38,A -85,B 0,C 180,E1 -4122.895,E2 -4122.895} C_VEL
LIN {X 0,Y 20.637,Z 1276.549,A -85,B 0,C 180,E1 -4132.119,E2 -4132.119} C_VEL
LIN {X 0,Y 13.973,Z 1276.737,A -85,B 0,C 180,E1 -4148.847,E2 -4148.847} C_VEL
LIN {X 0,Y 8.598,Z 1276.893,A -85,B 0,C 180,E1 -4186.69,E2 -4186.69} C_VEL
LIN {X 0,Y 7.736,Z 1276.915,A -85,B 0,C 180,E1 -4233.418,E2 -4233.418} C_VEL
LIN {X 0,Y 8.39,Z 1276.851,A -85,B 0,C 180,E1 -4253.558,E2 -4253.558} C_VEL
LIN {X 0,Y 22.404,Z 1276.386,A -85,B 0,C 180,E1 -4308.673,E2 -4308.673} C_VEL
LIN {X 0,Y 39.236,Z 1275.256,A -85,B 0,C 180,E1 -4319.587,E2 -4319.587} C_VEL
LIN {X 0,Y 15.982,Z 1276.733,A -85,B 0,C 180,E1 -4340.51,E2 -4340.51} C_VEL
LIN {X 0,Y 7.909,Z 1277.075,A -85,B 0,C 180,E1 -4402.947,E2 -4402.947} C_VEL
LIN {X 0,Y 10.584,Z 1276.898,A -85,B 0,C 180,E1 -4459.329,E2 -4459.329} C_VEL
LIN {X 0,Y 27.178,Z 1276.102,A -85,B 0,C 180,E1 -4493.917,E2 -4493.917} C_VEL
LIN {X 0,Y 39.325,Z 1275.23,A -85,B 0,C 180,E1 -4500.452,E2 -4500.452} C_VEL
LIN {X 0,Y 15.514,Z 1276.614,A -85,B 0,C 180,E1 -4522.75,E2 -4522.75} C_VEL
LIN {X 0,Y 7.935,Z 1276.895,A -85,B 0,C 180,E1 -4582.552,E2 -4582.552} C_VEL
LIN {X 0,Y 8.39,Z 1276.851,A -85,B 0,C 180,E1 -4613.558,E2 -4613.558} C_VEL
LIN {X 0,Y 9.219,Z 1278.851,A -85,B 0,C 180,E1 -4625.744,E2 -4625.744} C_VEL
LIN {X 0,Y 9.219,Z 1292,A -85,B 0,C 180,E1 -4625.744,E2 -4625.744} C_VEL
LIN {X 0,Y 9.219,Z 1292,A -85,B 0,C 180,E1 -4625.744,E2 -4625.744}

QRS_NEXT_CUT()

QRS_NEXT()
QRS_HOME()

END
